FUNCTION_BLOCK FB_HE_SATT_Sequence IMPLEMENTS I_HE_SATT_Sequence
VAR
    iFilterCombinationFinder : I_HE_SATT_FilterCombinationFinder;
    iFilterHolderSelector : I_HE_SATT_FilterHolderSelector;
    iPhotonEnergy_eV : I_HE_SATT_PhotonEnergy_eV;
    iFindOptimalFilterCombination : I_HE_SATT_FindOptimalFilterCombination;
    iFindOptimalThicknessFromFilterCombination : I_HE_SATT_FindOptimalThicknessFromFilterCombination;
    iCommands : I_HE_SATT_Commands;
    aiFilterHolder : REFERENCE TO ARRAY[1..PL_HE_SATT_Parameters.nNumHolders] OF I_HE_SATT_FilterHolder;

    eSequenceState : E_HE_SATT_SequenceState;
    
	fRequestedTransmission	: LREAL;
	eRequestedRoundingMode	: E_HE_SATT_RoundingMode;
	fRequestedAllowableTolerance	: LREAL;
    
    fbFilterCombinationCollector : FB_HE_SATT_FilterCombinationCollector;
    fbFilterCombinationCollectorDownselected : FB_HE_SATT_FilterCombinationCollector;
    
    iOptimalFilterCombination : I_HE_SATT_FilterCombination;
    
    afThickness : ARRAY[1..PL_HE_SATT_Parameters.nNumHolders] OF LREAL;
    
    nIteratorHolder : INT;
    iFilter : I_HE_SATT_Filter;
    
    bAllDone : BOOL;
END_VAR


IF iCommands.Reset THEN
    eSequenceState := E_HE_SATT_SequenceState.IDLE;
END_IF

CASE SequenceState OF
    E_HE_SATT_SequenceState.IDLE:
        // Do nothing for now
        
    E_HE_SATT_SequenceState.TRIGGER_DETERMINE_FILTER_COMBINATIONS:
        iFilterCombinationFinder.DetermineFilterCombinations(
            iFilterHolderSelector := iFilterHolderSelector,
            iFilterCombinationCollector := fbFilterCombinationCollector
        );
        
        eSequenceState := E_HE_SATT_SequenceState.CONFIRM_DETERMINE_FILTER_COMBINATIONS;
        
    E_HE_SATT_SequenceState.CONFIRM_DETERMINE_FILTER_COMBINATIONS:
        IF iFilterCombinationFinder.Status.bError THEN
            eSequenceState := E_HE_SATT_SequenceState.ERROR;
            // TODO: error handling
            RETURN;
        END_IF
        
        IF iFilterCombinationFinder.Status.bDone THEN
            eSequenceState := E_HE_SATT_SequenceState.TRIGGER_DOWNSELECT_FILTER_COMBINATIONS;
        END_IF
        
    E_HE_SATT_SequenceState.TRIGGER_DOWNSELECT_FILTER_COMBINATIONS:
        fbFilterCombinationCollector.DownselectByCouplingRule(
            iFilterHolderSelector := iFilterHolderSelector,
            iFilterCombinationCollector := fbFilterCombinationCollectorDownselected
        );
        
        eSequenceState := E_HE_SATT_SequenceState.CONFIRM_DOWNSELECT_FILTER_COMBINATIONS;
        
    E_HE_SATT_SequenceState.CONFIRM_DOWNSELECT_FILTER_COMBINATIONS:
        IF fbFilterCombinationCollector.DownselectStatus.bError THEN
            eSequenceState := E_HE_SATT_SequenceState.ERROR;
            // TODO: error handling
            RETURN;
        END_IF
        
        IF fbFilterCombinationCollector.DownselectStatus.bDone THEN
            eSequenceState := E_HE_SATT_SequenceState.TRIGGER_CALCULATE_OPTIMAL_FILTER_COMBINATION;
        END_IF
        
    E_HE_SATT_SequenceState.TRIGGER_CALCULATE_OPTIMAL_FILTER_COMBINATION:
        IF iPhotonEnergy_eV.Error THEN
            eSequenceState := E_HE_SATT_SequenceState.ERROR;
            // TODO: error handling
            RETURN;
        END_IF
    
        iFindOptimalFilterCombination.FindOptimalCombination(
            fPhotonEnergy_eV := iPhotonEnergy_eV.Value,
            fRequestedTransmission := fRequestedTransmission,
            eRequestedRoundingMode := eRequestedRoundingMode,
            fRequestedAllowableTolerance := fRequestedAllowableTolerance,
            iFilterCombinationCollector := fbFilterCombinationCollectorDownselected,
            iOptimalFilterCombination => iOptimalFilterCombination,
        );
        
        eSequenceState := E_HE_SATT_SequenceState.CONFIRM_CALCULATE_OPTIMAL_FILTER_COMBINATION;
        
    E_HE_SATT_SequenceState.CONFIRM_CALCULATE_OPTIMAL_FILTER_COMBINATION:
        IF iFindOptimalFilterCombination.Status.bError THEN
            eSequenceState := E_HE_SATT_SequenceState.ERROR;
            // TODO: error handling
            RETURN;
        END_IF
        
        IF iFindOptimalFilterCombination.Status.bDone THEN
            eSequenceState := E_HE_SATT_SequenceState.TRIGGER_CALCULATE_OPTIMAL_WEDGE_THICKNESSES;
        END_IF
        
    E_HE_SATT_SequenceState.TRIGGER_CALCULATE_OPTIMAL_WEDGE_THICKNESSES:
        IF iOptimalFilterCombination = 0 THEN
            eSequenceState := E_HE_SATT_SequenceState.ERROR;
            // TODO: error handling
            RETURN;
        END_IF
        
        IF iPhotonEnergy_eV.Error THEN
            eSequenceState := E_HE_SATT_SequenceState.ERROR;
            // TODO: error handling
            RETURN;
        END_IF
        
        iFindOptimalThicknessFromFilterCombination.FindOptimalThicknessFromFilterCombination(
            fPhotonEnergy_eV := iPhotonEnergy_eV.Value,
            fRequestedTransmission := fRequestedTransmission,
            iFilterCombination := iOptimalFilterCombination,
            afThickness => afThickness
        );
        
    E_HE_SATT_SequenceState.CONFIRM_CALCULATE_OPTIMAL_WEDGE_THICKNESSES:
        IF iFindOptimalThicknessFromFilterCombination.Status.bError THEN
            eSequenceState := E_HE_SATT_SequenceState.ERROR;
            // TODO: error handling
            RETURN;
        END_IF
        
        IF iFindOptimalThicknessFromFilterCombination.Status.bDone THEN
            eSequenceState := E_HE_SATT_SequenceState.CONFIRM_MOVE_PERMITTED;
        END_IF
        
    E_HE_SATT_SequenceState.CONFIRM_MOVE_PERMITTED:
        IF iCommands.PermitMove THEN
            eSequenceState := E_HE_SATT_SequenceState.TRIGGER_MOVE_START;
        END_IF
        
    E_HE_SATT_SequenceState.TRIGGER_MOVE_START:
        FOR nIteratorHolder := 1 TO PL_HE_SATT_Parameters.nNumHolders BY 1 DO
            iFilter := iOptimalFilterCombination.GetFilter(nIteratorHolder);
            
            aiFilterHolder[nIteratorHolder].MoveToFilter(
                iFilter := iFilter,
                fThickness := afThickness[nIteratorHolder]
            );
        END_FOR
        
        eSequenceState := E_HE_SATT_SequenceState.CONFIRM_MOVE_COMPLETE;
        
    E_HE_SATT_SequenceState.CONFIRM_MOVE_COMPLETE:
        FOR nIteratorHolder := 1 TO PL_HE_SATT_Parameters.nNumHolders BY 1 DO
            IF aiFilterHolder[nIteratorHolder].Status.bError THEN
                eSequenceState := E_HE_SATT_SequenceState.ERROR;
                // TODO: error handling
                RETURN;
            END_IF
        END_FOR
        
        bAllDone := TRUE;
        
        FOR nIteratorHolder := 1 TO PL_HE_SATT_Parameters.nNumHolders BY 1 DO
            bAllDone := bAllDone AND aiFilterHolder[nIteratorHolder].Status.bDone;
        END_FOR
        
        IF bAllDone THEN
            eSequenceState := E_HE_SATT_SequenceState.IDLE;
            // TODO: lof successful completion of move.
        END_IF
        
    E_HE_SATT_SequenceState.ERROR:
        // TODO: error handling
        
END_CASE


METHOD FB_Init: BOOL
VAR_INPUT
    bInitRetains: BOOL; // TRUE: the retain variables are initialized (reset warm / reset cold)
    bInCopyCode: BOOL;  // TRUE: the instance will be copied to the copy code afterward (online change)   
    
    iFilterCombinationFinder : I_HE_SATT_FilterCombinationFinder;
    iFilterHolderSelector : I_HE_SATT_FilterHolderSelector;
    iFindOptimalFilterCombination : I_HE_SATT_FindOptimalFilterCombination;
    iPhotonEnergy_eV : I_HE_SATT_PhotonEnergy_eV;
    iCommands : I_HE_SATT_Commands;
    aiFilterHolder : REFERENCE TO ARRAY[1..PL_HE_SATT_Parameters.nNumHolders] OF I_HE_SATT_FilterHolder;
END_VAR

THIS^.iFilterCombinationFinder := iFilterCombinationFinder;
THIS^.iFilterHolderSelector := iFilterHolderSelector;
THIS^.iFindOptimalFilterCombination := iFindOptimalFilterCombination;
THIS^.iPhotonEnergy_eV := iPhotonEnergy_eV;
THIS^.iCommands := iCommands;
THIS^.aiFilterHolder REf= aiFilterHolder;
END_METHOD

PROPERTY PUBLIC SequenceState : E_HE_SATT_SequenceState
GET

SequenceState := THIS^.eSequenceState;
END_GET
END_PROPERTY


METHOD Start
VAR_INPUT
	(* [0.0 - 1.0]*)
	fRequestedTransmission	: LREAL;
	eRequestedRoundingMode	: E_HE_SATT_RoundingMode;
	fRequestedAllowableTolerance	: LREAL;
END_VAR

THIS^.fRequestedTransmission := fRequestedTransmission;
THIS^.eRequestedRoundingMode := eRequestedRoundingMode;
THIS^.fRequestedAllowableTolerance := fRequestedAllowableTolerance;

THIS^.eSequenceState := E_HE_SATT_SequenceState.TRIGGER_DETERMINE_FILTER_COMBINATIONS;
END_METHOD

END_FUNCTION_BLOCK

(* stored: Version 1.1.0.1
   POU FB_HE_SATT_Sequence: Id {dfc1a105-47c7-4948-b3e0-930059e1be08}, SpecialFunc None
   Method FB_Init: Id {f4d7ec53-0767-47c2-8c9e-bc2f05fb3bef}
   Property SequenceState: Id {929427a0-ccc7-4946-99ca-5deed82b5dcf}
   Get Get: Id {6ccd5faf-c46b-4e55-9e3a-0a24258f6c4b}
   Method Start: Id {f4fa7a48-3d5a-4228-b11a-aed8bb01baf1} *)
